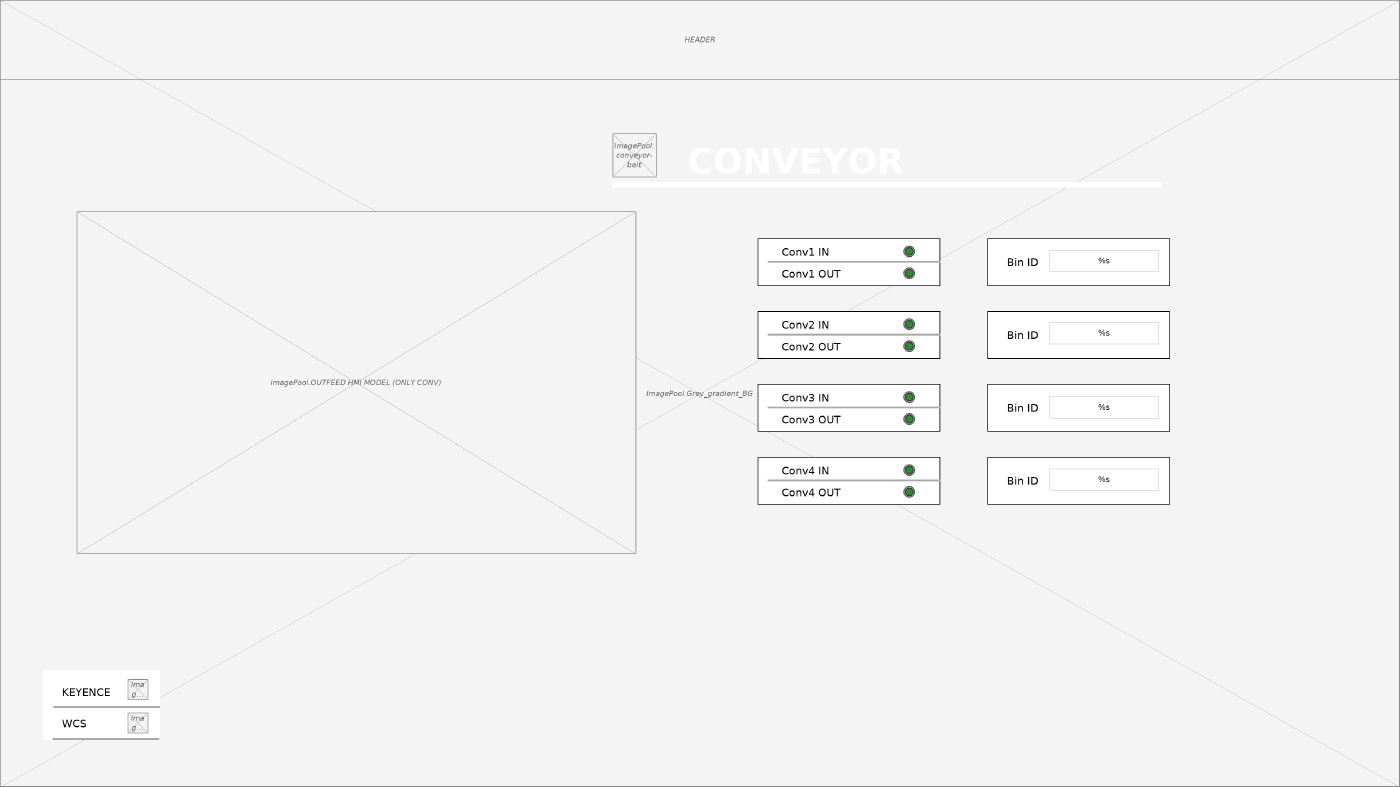
VISUALIZATION CONVEYOR_PAGE  // 1920x1080
    Image (0,0 1920x1080), image: ImagePool.Grey_gradient_BG
    Frame (0,0 1920x109)
        shows HEADER()
    Image (105,290 767x470), image: ImagePool.OUTFEED HMI MODEL (ONLY CONV)
    Rectangle (885,184 413x74), "CONVEYOR"
    Rectangle (840,250 752x7)
    Image (840,183 60x60), image: ImagePool.conveyor-belt
    Group (1039,327 250x365)
        Group (0,0 250x65)
            RoundedRectangle (0,0 250x65)
            Rectangle (30,4 118x30), "Conv1 IN"
            Rectangle (30,34 118x30), "Conv1 OUT"
            Lamp1 (199,9 18x18), variable: IO.bConv1_In, style: Lamp-Lamp1-Green
            Lamp1 (199,39 18x18), variable: IO.bConv1_Out, style: Lamp-Lamp1-Green
            Rectangle (14,31 236x2)
        Group (0,100 250x65)
            RoundedRectangle (0,0 250x65)
            Rectangle (30,4 118x30), "Conv2 IN"
            Rectangle (30,34 118x30), "Conv2 OUT"
            Lamp1 (199,9 18x18), variable: IO.bConv2_In, style: Lamp-Lamp1-Green
            Lamp1 (199,39 18x18), variable: IO.bConv2_Out, style: Lamp-Lamp1-Green
            Rectangle (14,31 236x2)
        Group (0,200 250x65)
            RoundedRectangle (0,0 250x65)
            Rectangle (30,4 118x30), "Conv3 IN"
            Rectangle (30,34 118x30), "Conv3 OUT"
            Lamp1 (199,9 18x18), variable: IO.bConv3_In, style: Lamp-Lamp1-Green
            Lamp1 (199,39 18x18), variable: IO.bConv3_Out, style: Lamp-Lamp1-Green
            Rectangle (14,31 236x2)
        Group (0,300 250x65)
            RoundedRectangle (0,0 250x65)
            Rectangle (30,4 118x30), "Conv4 IN"
            Rectangle (30,34 118x30), "Conv4 OUT"
            Lamp1 (199,9 18x18), variable: IO.bConv4_In, style: Lamp-Lamp1-Green
            Lamp1 (199,39 18x18), variable: IO.bConv4_Out, style: Lamp-Lamp1-Green
            Rectangle (14,31 236x2)
    Group (59,920 160x95)
        RoundedRectangle (0,0 160x95)
        RoundedRectangle (23,21 109x18), "KEYENCE"
        RoundedRectangle (23,64 92x18), "WCS"
        Rectangle (14,49 146x2)
        Rectangle (13,93 146x2)
        Image (116,12 28x28), invisible if: IO.fbClient_QR.bConnected, image: ImagePool.no-wifi
        Image (116,12 28x28), invisible if: NOT IO.fbClient_QR.bConnected, image: ImagePool.wifi
        Image (116,58 28x28), invisible if: IO.fbClient_ASRS.bConnected, image: ImagePool.no-wifi
        Image (116,58 28x28), invisible if: NOT IO.fbClient_ASRS.bConnected, image: ImagePool.wifi
    Group (1354,327 250x65)
        RoundedRectangle (0,0 250x65)
        Rectangle (24,18 118x30), "Bin ID"
    Group (1354,427 250x65)
        RoundedRectangle (0,0 250x65)
        Rectangle (24,18 118x30), "Bin ID"
    Group (1354,527 250x65)
        RoundedRectangle (0,0 250x65)
        Rectangle (24,18 118x30), "Bin ID"
    Group (1354,627 250x65)
        RoundedRectangle (0,0 250x65)
        Rectangle (24,18 118x30), "Bin ID"
    Textfield (1439,343 150x30), "%s", text variable: IO.abinID_Set[2]
    Textfield (1439,442 150x30), "%s", text variable: IO.abinID_Set[4]
    Textfield (1439,544 150x30), "%s", text variable: IO.abinID_Set[6]
    Textfield (1439,643 150x30), "%s", text variable: IO.abinID_Set[8]
END_VISUALIZATION

(* stored: Version 1.1.0.1, ProductVersion 3.1.4024.12
   Visu CONVEYOR_PAGE: Id {74d67950-ef01-402a-8eba-6cb9b71b927b} *)
